// TIA Portal V18 export
DATA_BLOCK "PartDataManage_Part1_DB"   // DB1501
VERSION : 0.1
// stored: AutoNumber true, DBAccessibleFromOPCUA true, DBAccessibleFromWebserver true, InstanceOfName PartDataManage, InstanceOfType FB
"PartDataManage"
   // VAR_INPUT
   //    iReset : Bool;
   //    iScannerTrigger : Bool;
   //    iStringRecived : String;
   //    iMaterialType : String;
   //    iSaveToBuffer : Bool;
   //    iCodeType : Bool;
   //    iDecrementCnt : DInt;
   //    iDecrementTrigger : Bool;
   //    iBufferBoxes : Int;
   // END_VAR
   // VAR_IN_OUT
   //    ioMaterialActive : Bool;
   //    io_MaterialManage : "PartData_UDT";
   // END_VAR
   // VAR
   //    NO : Array[0..6] of Int;
   //    sString_MId : String;
   //    sKeyChar : Char;
   //    Puls : Array[0..20] of Bool;
   //    R_TRIG_MaterialActive { S7_SetPoint := 'True'} : R_TRIG;
   //    R_TRIG_ScannerTrigger { S7_SetPoint := 'True'} : R_TRIG;
   //    IEC_Timer_MaterialActive { S7_SetPoint := 'True'} : TON_TIME;
   //    R_TRIG_DecrementTrigger { S7_SetPoint := 'True'} : R_TRIG;
   //    "R_TRIG_PartQuality+1" { S7_SetPoint := 'True'} : R_TRIG;
   //    "R_TRIG_PartQuality-1" { S7_SetPoint := 'True'} : R_TRIG;
   //    R_TRIG_ClearCurrentBox { S7_SetPoint := 'True'} : R_TRIG;
   //    R_TRIG_ClearAllBox { S7_SetPoint := 'True'} : R_TRIG;
   //    R_TRIG_SaveToBuffer { S7_SetPoint := 'True'} : R_TRIG;
   //    Timer_PartQualityAckPB { S7_SetPoint := 'True'} : TON_TIME;
   // END_VAR
BEGIN
END_DATA_BLOCK
